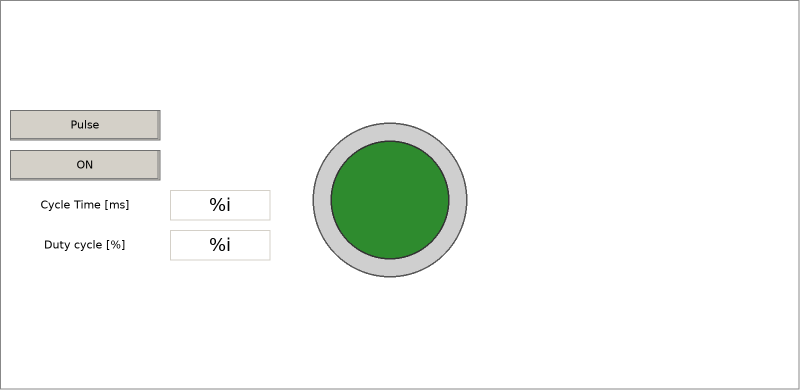
VISUALIZATION VisuPWMControl  // 800x390
VAR_IN_OUT
	pDev : POINTER TO FB_DevPWMGenerator;
END_VAR
    Lamp1 (300,110 180x180), variable: pDev^.qbOutput, style: Lamp-Lamp1-Green
    Button (10,110 150x30), "Pulse"
        toggle pDev^.bCmdPWMCycle
    Button (10,150 150x30), "ON"
        tap pDev^.bCmdOn
    Textfield (170,190 100x30), "%i", text variable: pDev^.nPeriodLength
        OnMouseUp: write the text variable via VisuDialogs.Numpad
    Label (10,190 150x30), "Cycle Time [ms]"
    Label (10,230 150x30), "Duty cycle [%]"
    Textfield (170,230 100x30), "%i", text variable: pDev^.nDutyCycle
        OnMouseClick: write the text variable via VisuDialogs.Numpad, min 0, max 100
END_VISUALIZATION

(* stored: Version 1.1.0.1, ProductVersion 3.1.4024.11
   Visu VisuPWMControl: Id {15593216-3553-0239-0441-986775d919de} *)
